FUNCTION Convert_LINT_TO_BYTE : Hresult
VAR_INPUT
	in : LINT;
	out : REFERENCE TO BYTE;
END_VAR
VAR
	converted : BYTE;
END_VAR

converted := LINT_TO_BYTE(in);

IF (BYTE_TO_LINT(converted) <> in) THEN
	Convert_LINT_TO_BYTE := INCOMPATIBLE;
	RETURN;
END_IF

out := converted;

END_FUNCTION

(* stored: Version 1.1.0.1, ProductVersion 3.1.4024.12
   POU Convert_LINT_TO_BYTE: Id {841795fd-da00-4369-94bb-9dd2d65d5c75}, SpecialFunc None *)
